	#StB_Hi := #IUDT_Analog_In.IBt_Enable_ControlLevel[1] AND #Level_Control_HoLo.QB_Hi;
	#StB_Hi_Q := #Level_Control_HoLo.QB_Hi AND #IUDT_Analog_In.IBt_Block_ControlLevel[1];
	#QB_Hi_Alarm := #StB_Hi_Q;
	
	#StB_Lo := #IUDT_Analog_In.IBt_Enable_ControlLevel[2] AND #Level_Control_HoLo.QB_Lo;
	#StB_Lo_Q :=  #Level_Control_HoLo.QB_Lo AND #IUDT_Analog_In.IBt_Block_ControlLevel[2];
	#QB_Lo_Alarm := #StB_Lo_Q;
	
	#StB_LoLo := (#StB_LoLo AND NOT #TmB_Reset_Bit)
	OR #IUDT_Analog_In.IBt_Enable_ControlLevel[3] AND #Level_Control_HoLo.QB_LoLo;
	#StB_LoLo_Q := (#StB_LoLo_Q AND NOT #TmB_Reset_Bit)
	OR #Level_Control_HoLo.QB_LoLo AND #IUDT_Analog_In.IBt_Block_ControlLevel[3];
	#QB_LoLo_Fault := #StB_LoLo_Q;
	
	
	
	//IWCword
	#IUDT_Analog_In.IW_CTW[0] := False;
	
	//Word of State
	//Fault
	#IUDT_Analog_In.QW_STW[0] := #StB_HiHi OR #StB_LoLo OR #TmB_Sensor_In_Zero OR #StB_PowerFault;
	// Alarm
	#IUDT_Analog_In.QW_STW[1] := #StB_Hi OR #StB_Lo;
	// All OK
	#IUDT_Analog_In.QW_STW[2] := NOT #IUDT_Analog_In.QW_STW[0] AND NOT #IUDT_Analog_In.QW_STW[1];
	#IUDT_Analog_In.QW_STW[3] := #TmB_Sensor_In_Zero AND (( #IB_PowerControl AND #IB_EnablePowerControl) OR NOT #IB_EnablePowerControl );
	#IUDT_Analog_In.QW_STW[4] := #StB_HiHi;
	#IUDT_Analog_In.QW_STW[5] := #StB_Hi;
	#IUDT_Analog_In.QW_STW[6] := #StB_Lo;
	#IUDT_Analog_In.QW_STW[7] := #StB_LoLo;
	
	#IUDT_Analog_In.QW_STW[9] := #TmB_Reset_Bit;
	#IUDT_Analog_In.QW_STW[10] := #StB_PowerFault;
	#IUDT_Analog_In.QW_STW[11] := #IB_PowerControl;
	
	//Word of Alarm and fault
	#IUDT_Analog_In.QDW_Message[0] := #TmB_Sensor_In_Zero;
	#IUDT_Analog_In.QDW_Message[1] := #StB_HiHi;
	#IUDT_Analog_In.QDW_Message[2] := #StB_LoLo;
	#IUDT_Analog_In.QDW_Message[3] := #StB_PowerFault;
	
	#IUDT_Analog_In.QDW_Message[14] := #StB_Hi;
	#IUDT_Analog_In.QDW_Message[15] := #StB_Lo;
	
	#IUDT_Analog_In.QDW_Message[16] := #IUDT_Analog_In.QW_STW[8];
	
	#QW_STW := #IUDT_Analog_In.QW_STW;
	
	
END_FUNCTION_BLOCK

FUNCTION_BLOCK "Level_Control_HoLo"
{ S7_Optimized_Access := 'FALSE' }
VERSION : 0.1
   VAR_INPUT 
      IB_Enable_Func : Bool;
      IDW_Actual_Value : Real;
      IDW_Set_HiHi : Real;
      IDW_Set_Hi : Real;
      IDW_Set_LoLo : Real;
      IDW_Set_Lo : Real;
      IW_Time_HiHi : Int;
      IW_Time_Hi : Int;
      IW_Time_LoLo : Int;
      IW_Time_Lo : Int;
   END_VAR

   VAR_OUTPUT 
      QB_HiHi : Bool;
      QB_Hi : Bool;
      QB_LoLo : Bool;
      QB_Lo : Bool;
   END_VAR

   VAR 
      Timer_TON_HiHi {InstructionName := 'TON'; LibVersion := '1.0'} : TON;
      Timer_TON_Hi {InstructionName := 'TON'; LibVersion := '1.0'} : TON;
      Timer_TON_LoLo {InstructionName := 'TON'; LibVersion := '1.0'} : TON;
      Timer_TON_Lo {InstructionName := 'TON'; LibVersion := '1.0'} : TON;
   END_VAR

   VAR_TEMP 
      Tm_Time_HI : DInt;
      Tm_Time_Lo : DInt;
      Tm_Time_HIHI : DInt;
      Tm_Time_LOLO : DInt;
   END_VAR


BEGIN
	//Hi
	#Tm_Time_HI := INT_TO_DINT(#IW_Time_Hi);
	#Timer_TON_Hi(IN := #IDW_Actual_Value > #IDW_Set_Hi AND #IB_Enable_Func AND #IDW_Set_Hi <> 0,
	              PT := DINT_TO_TIME(#Tm_Time_HI * 1000),
	              
	              Q => #QB_Hi);
	
	//HiHi
	#Tm_Time_HIHI := INT_TO_DINT(#IW_Time_HiHi);
	#Timer_TON_HiHi(IN := #IDW_Actual_Value > #IDW_Set_HiHi AND #IB_Enable_Func AND #IDW_Set_HiHi <> 0,
	                PT := DINT_TO_TIME(#Tm_Time_HIHI * 1000),
	                Q => #QB_HiHi);
	//Lo
	#Tm_Time_Lo := INT_TO_DINT(#IW_Time_Lo);
	#Timer_TON_Lo(IN := #IDW_Actual_Value < #IDW_Set_Lo AND #IB_Enable_Func AND #IDW_Set_Lo <> 0,
	              PT := DINT_TO_TIME(#Tm_Time_Lo * 1000),
	              Q => #QB_Lo);
	//LoLo
	#Tm_Time_LOLO := INT_TO_DINT(#IW_Time_LoLo);
	#Timer_TON_LoLo(IN := #IDW_Actual_Value < #IDW_Set_LoLo AND #IB_Enable_Func AND #IDW_Set_LoLo <> 0,
	                PT := DINT_TO_TIME(#Tm_Time_LOLO * 1000),
	                Q => #QB_LoLo);
END_FUNCTION_BLOCK

FUNCTION_BLOCK "Smoothing"
{ S7_Optimized_Access := 'FALSE' }
VERSION : 0.1
   VAR_INPUT 
      IDW_Input_Value : Real;
      IW_Time_Smoothing : Int;
      IB_Gen_In : Bool;
      IW_Gen_Value : DInt;
   END_VAR

   VAR_OUTPUT 
      QDW_Smoothing_Value : Real;
   END_VAR

   VAR 
      Value_array : Array[0..100] of Real;
      St_PointArray : Int;
      St_Counter : Int;
      St_Counter_Shift : Int;
      St_Counter_Summ : Int;
      St_Summ_Arr : Real;
   END_VAR

   VAR_TEMP 
      Temp_UDint : DInt;
   END_VAR


BEGIN
	#Temp_UDint := #IW_Time_Smoothing;
	IF #IW_Time_Smoothing>0 THEN
	        
	    #St_PointArray := (DINT_TO_INT((#Temp_UDint * 100) / #IW_Gen_Value));
	    IF #St_PointArray>100
	    THEN
	        #St_PointArray := 100;
	    END_IF;
	    
	    //#R_TRIG_Instance(CLK:=#IB_Gen_In);
	    
	    IF #IB_Gen_In THEN
	        
	        #St_Summ_Arr := 0;
	        FOR #St_Counter_Shift := #St_PointArray  TO 2 BY -1 DO
	            #Value_array[#St_Counter_Shift] := #Value_array[#St_Counter_Shift - 1];
	        END_FOR;
	        #Value_array[1] := #IDW_Input_Value;
	        //Обмеження лічильника
	        IF #St_Counter<#St_PointArray THEN
	            #St_Counter := #St_Counter + 1;
	        ELSE
	            #St_Counter := #St_PointArray;
	        END_IF;
	        //Сумування масиву
	        FOR #St_Counter_Summ := 1 TO #St_Counter DO
	            #St_Summ_Arr := #St_Summ_Arr + #Value_array[#St_Counter_Summ];
	        END_FOR;
	        //Усереднене значення масиву
	        #QDW_Smoothing_Value := #St_Summ_Arr / (#St_Counter);
	    END_IF;
	    
	ELSE
	#QDW_Smoothing_Value := #IDW_Input_Value;
	#St_Counter := 0;
	END_IF;
	
	
	
	
END_FUNCTION_BLOCK

FUNCTION "Scaling_TSS" : Void
{ S7_Optimized_Access := 'FALSE' }
VERSION : 0.1
   VAR_INPUT 
      In_Value : Real;
      In_Max : Real;
      In_Min : Real;
      Out_Max : Real;
      Out_Min : Real;
   END_VAR

   VAR_OUTPUT 
      Out_Value : Real;
      Fault : Bool;
      Senser_In_Zero : Bool;
   END_VAR

   VAR_TEMP 
      Diap_In : Real;
      Diap_Out : Real;
      In_prop : Real;
      Out_prop_1 : Real;
      Value_Out : Real;
      Value_IN : Real;
      Temp_Sensor_In_Zero : Bool;
   END_VAR


BEGIN
	#Diap_In := #In_Max - #In_Min;
	#Diap_Out := #Out_Max - #Out_Min;
	#Value_IN := #In_Value - #In_Min;
	IF #In_Max < #In_Min                                   //Перевірка чи максимальні значення не менші мінімальних
	    OR (#Out_Max < #Out_Min)                         //якщо так то помилка 
	THEN
	    #Fault := true;
	    
	ELSE
	    //Перевірка чи апаратне значення не за доступними межами; якщо так то датчик в нулі
	    // IF #In_Value = 32768
	    //     OR (#In_Value = -32768)
	    // THEN
	    //     #Senser_In_Zero := true;
	    //     #Temp_Sensor_In_Zero := true;
	    //     #Out_Value := 0;
	    // ELSE
	    //     #Senser_In_Zero := false;
	    //     #Temp_Sensor_In_Zero := false;
	    // END_IF;
	    
	    #Fault := false;
	    #In_prop := (#Value_IN * 100) / #Diap_In;                    //Вхід в процентах
	    #Out_prop_1 := (#Diap_Out * 1) / 100;                       //1 процент від шкали виходу
	    #Value_Out := #In_prop * #Out_prop_1;                       //Вихід в процентах    
	    
	    IF #In_Value > #In_Max
	        // AND NOT (#Temp_Sensor_In_Zero)
	    THEN
	        #Out_Value := #Out_Max;
	    ELSIF #In_Value < #In_Min
	        // AND NOT (#Temp_Sensor_In_Zero)
	    THEN
	        #Out_Value := #Out_Min;
	    ELSIF #In_Value >= #In_Min AND #In_Value <= #In_Max
	        // AND NOT #Temp_Sensor_In_Zero
	    THEN
	        #Out_Value := #Out_Min + #Value_Out;
	    END_IF;
	    
	    
	END_IF;
	
	
	
	
	
END_FUNCTION
